(* Logix 5000 project; controller Sucrose_Main Emulate 5570 rev 20.12; software revision 20.01; part 8 of 30 *)
(* tags used below, declared in another part *)
   AI_E23_0 : REAL[8];   // Analog Input EN2T_FLX 192.168.1.23
   AI_E23_1 : REAL[8];   // Analog Input EN2T_FLX 192.168.1.23
   Alarm_ACK_Master_Timer : TIMER;
   ClearFault_Master : BOOL;
   DI_E20_0 : ALIAS FOR FLX_E20:0:I;   // Discrete Input EN2T_FLX 192.168.1.20
   DI_E20_2 : ALIAS FOR FLX_E20:2:I;   // Discrete Input EN2T_FLX 192.168.1.20
   DISCHARGE_NO_ALARM : BOOL;   // SUCROSE HEADER NO ACTIVE ALARMS FOR P_23_01_01 PATH
   DISCHARGE_NO_ALARM2 : BOOL;   // SUCROSE HEADER NO ACTIVE ALARMS FOR P_23_01_02 PATH
   DO_E20_3 : ALIAS FOR FLX_E20:3:O;   // Discrete Output EN2T_FLX 192.168.1.20
   FV230411_AOI : QSI_Flow_Valve;   // FV-23-04-11-O SUCROSE TANK #1 TO TRANSFER PUMP #1 MIX PROOF VALVE OPEN
   FV230441_AOI : QSI_Flow_Valve;   // FV-23-04-41-O SUCROSE TRANSFER PUMP #1 DISCHARGE TO FILTRATRION MIX PROOF VALVE OPEN
   FV230442_AOI : QSI_Flow_Valve;   // FV-23-04-42-O SUCROSE TRANSFER PUMP #2 DISCHARGE TO FILTRATRION MIX PROOF VALVE OPEN
   HEADER_LOW_FLOW : DINT;
   ONESHOTBITS : INT[10];
   P230401_AOI : PF525_VFD_E_ENET;   // P-23-04-01 SUCROSE TRANSFER PUMP 1
   P230402_AOI : PF525_VFD_E_ENET;   // P-23-04-02 SUCROSE TRANSFER PUMP 2
   P620101_AOI : PF525_VFD_E_ENET;   // P-62-01-01 CIP RETURN UP
   Rung_Comment : BOOL;
   SUCROSE_HEADER_NO_ALARM : BOOL;
   SUCROSE_HEADER_WATER_PURGE_GALLONS_TOTAL : DINT;
   SUCROSE_HEADER_WATER_PURGE_SP : DINT;
   Sucrose_MM_Enable : BOOL;
   SUCROSE_TANK_QUEUE_LEVEL : DINT;
   SucroseCIP_P230401_REMOTE : CIP_REMOTE;
   SucroseCIP_P230402_REMOTE : CIP_REMOTE;
   SucroseCIP_RINGMAIN_REMOTE : CIP_REMOTE;
   SucroseCIP_TK230101_REMOTE : CIP_REMOTE;
   SucroseCIP_TK230201_REMOTE : CIP_REMOTE;
   SucroseCIP_TK230301_REMOTE : CIP_REMOTE;
   SucroseDischarge : Area_Program;
   SucroseFiltration : Area_Program;
   SucroseTanks : Area_Program;
   SUROSE_HEADER_WATER_PURGE_GALS_PER_SEC : DINT;
   TK_23_01_01_LOW_LEVEL : DINT;
   TK_23_02_01_LOW_LEVEL : DINT;
   TK_23_03_01_LOW_LEVEL : DINT;
(* CIP_RemoteArea_EN2T_IO_Discrete_DO_E25_5, continued *)

ROUTINE MainRoutine   (* ladder *)
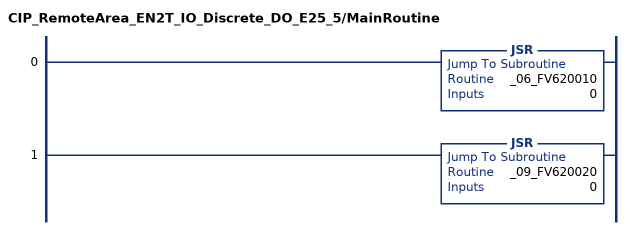
   0: JSR(_06_FV620010,0);
   1: JSR(_09_FV620020,0);
END_ROUTINE
END_PROGRAM

PROGRAM CIP_RemoteArea_EN2T_IO_Drives   (* main routine MainRoutine *)

ROUTINE E32_P620101   (* ladder *)
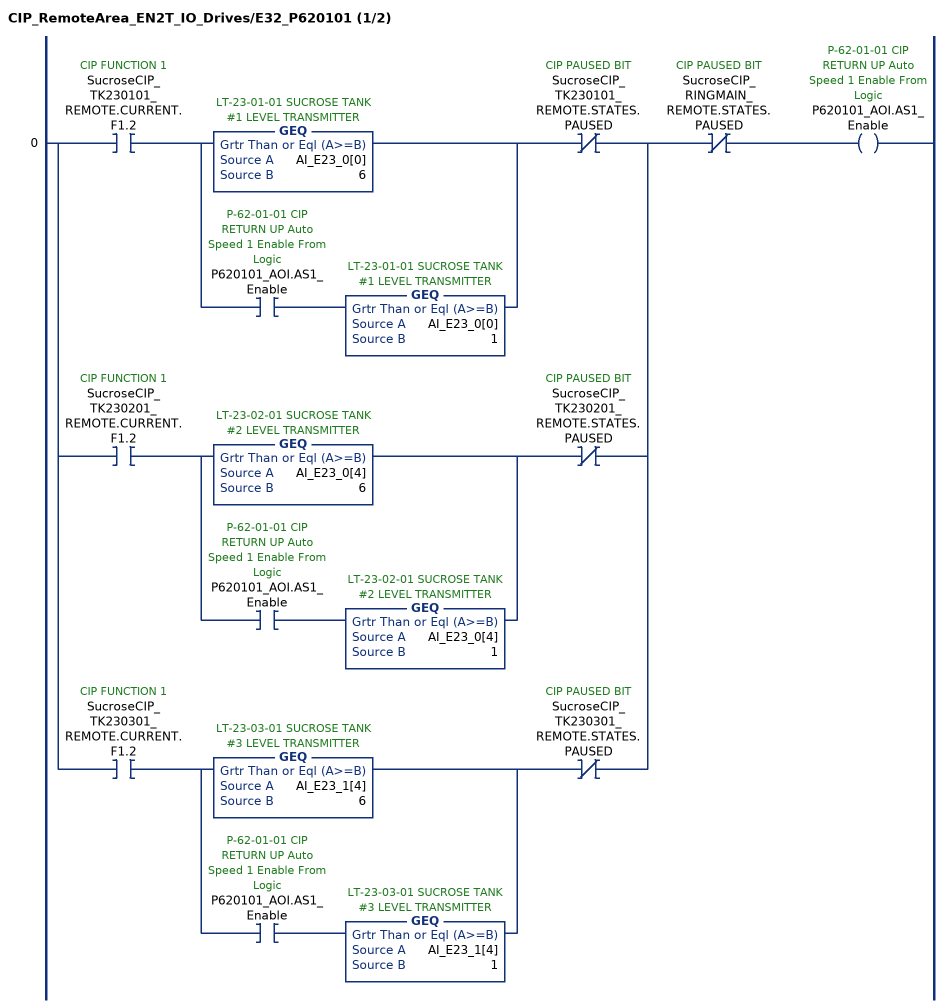
   0: [XIC(SucroseCIP_TK230101_REMOTE.CURRENT.F1.2) [GEQ(AI_E23_0[0],6) ,XIC(P620101_AOI.AS1_Enable) GEQ(AI_E23_0[0],1) ] XIO(SucroseCIP_TK230101_REMOTE.STATES.PAUSED) ,XIC(SucroseCIP_TK230201_REMOTE.CURRENT.F1.2) [GEQ(AI_E23_0[4],6) ,XIC(P620101_AOI.AS1_Enable) GEQ(AI_E23_0[4],1) ] XIO(SucroseCIP_TK230201_REMOTE.STATES.PAUSED) ,XIC(SucroseCIP_TK230301_REMOTE.CURRENT.F1.2) [GEQ(AI_E23_1[4],6) ,XIC(P620101_AOI.AS1_Enable) GEQ(AI_E23_1[4],1) ] XIO(SucroseCIP_TK230301_REMOTE.STATES.PAUSED) ]XIO(SucroseCIP_RINGMAIN_REMOTE.STATES.PAUSED)OTE(P620101_AOI.AS1_Enable);
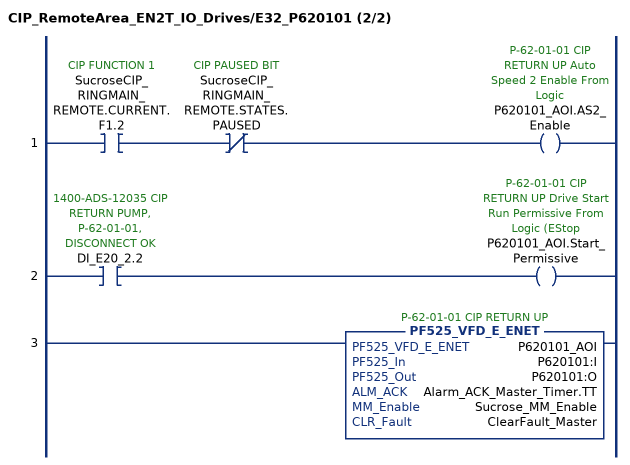
   1: XIC(SucroseCIP_RINGMAIN_REMOTE.CURRENT.F1.2)XIO(SucroseCIP_RINGMAIN_REMOTE.STATES.PAUSED)OTE(P620101_AOI.AS2_Enable);
   2: XIC(DI_E20_2.2)OTE(P620101_AOI.Start_Permissive);
   3: PF525_VFD_E_ENET(P620101_AOI,P620101:I,P620101:O,Alarm_ACK_Master_Timer.TT,Sucrose_MM_Enable,ClearFault_Master);
END_ROUTINE

ROUTINE MainRoutine   (* ladder *)
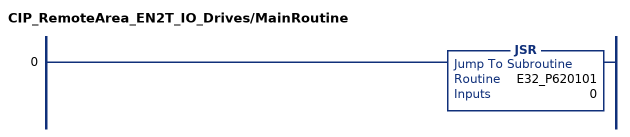
   0: JSR(E32_P620101,0);
END_ROUTINE
END_PROGRAM

PROGRAM DischargeArea_AutoLogic   (* main routine MainRoutine *)
VAR
   HEADER_HIGH_PRESSUR : DINT;
   HEADER_LOW_PRESSUR : DINT;
END_VAR

ROUTINE Alarm_Logic   (* ladder *)
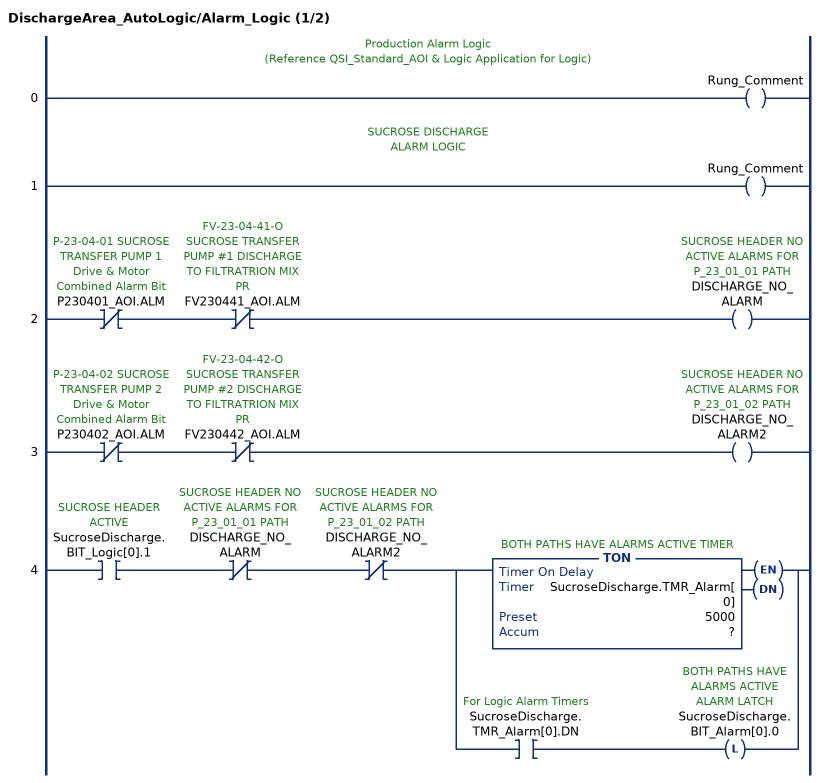
   // Production Alarm Logic
   // (Reference QSI_Standard_AOI & Logic Application for Logic)
   0: OTE(Rung_Comment);
   // SUCROSE DISCHARGE
   // ALARM LOGIC
   1: OTE(Rung_Comment);
   2: XIO(P230401_AOI.ALM)XIO(FV230441_AOI.ALM)OTE(DISCHARGE_NO_ALARM);
   3: XIO(P230402_AOI.ALM)XIO(FV230442_AOI.ALM)OTE(DISCHARGE_NO_ALARM2);
   4: XIC(SucroseDischarge.BIT_Logic[0].1)XIO(DISCHARGE_NO_ALARM)XIO(DISCHARGE_NO_ALARM2)[TON(SucroseDischarge.TMR_Alarm[0],?,?) ,XIC(SucroseDischarge.TMR_Alarm[0].DN) OTL(SucroseDischarge.BIT_Alarm[0].0) ];
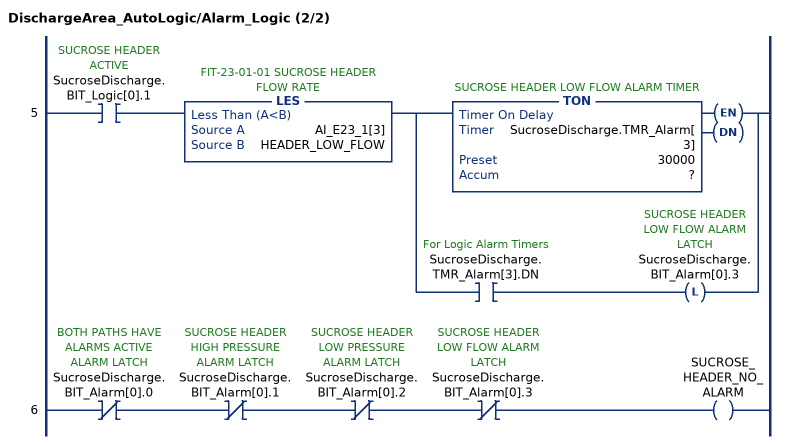
   5: XIC(SucroseDischarge.BIT_Logic[0].1)LES(AI_E23_1[3],HEADER_LOW_FLOW)[TON(SucroseDischarge.TMR_Alarm[3],?,?) ,XIC(SucroseDischarge.TMR_Alarm[3].DN) OTL(SucroseDischarge.BIT_Alarm[0].3) ];
   6: XIO(SucroseDischarge.BIT_Alarm[0].0)XIO(SucroseDischarge.BIT_Alarm[0].1)XIO(SucroseDischarge.BIT_Alarm[0].2)XIO(SucroseDischarge.BIT_Alarm[0].3)OTE(SUCROSE_HEADER_NO_ALARM);
END_ROUTINE

ROUTINE Control_Logic   (* ladder *)
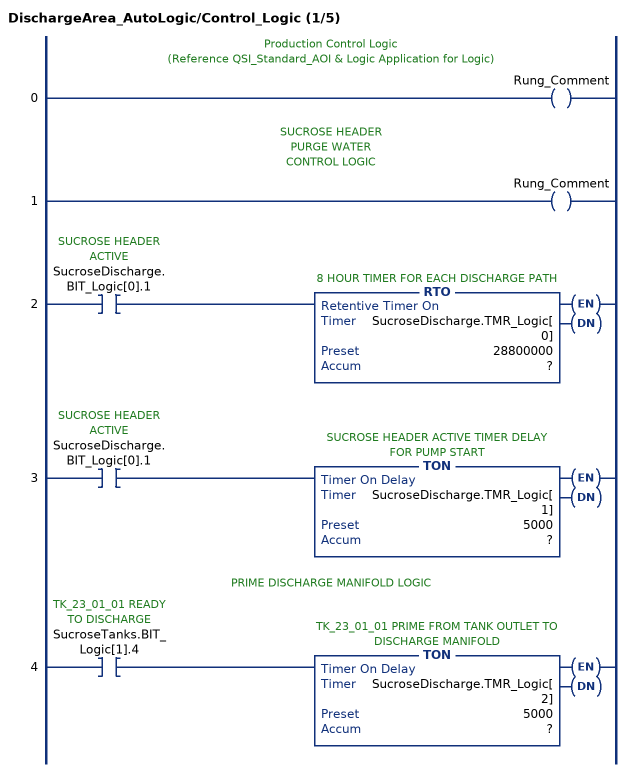
   // Production Control Logic
   // (Reference QSI_Standard_AOI & Logic Application for Logic)
   0: OTE(Rung_Comment);
   // SUCROSE HEADER
   // PURGE WATER
   // CONTROL LOGIC
   1: OTE(Rung_Comment);
   2: XIC(SucroseDischarge.BIT_Logic[0].1)RTO(SucroseDischarge.TMR_Logic[0],?,?);
   3: XIC(SucroseDischarge.BIT_Logic[0].1)TON(SucroseDischarge.TMR_Logic[1],?,?);
   // PRIME DISCHARGE MANIFOLD LOGIC
   4: XIC(SucroseTanks.BIT_Logic[1].4)TON(SucroseDischarge.TMR_Logic[2],?,?);
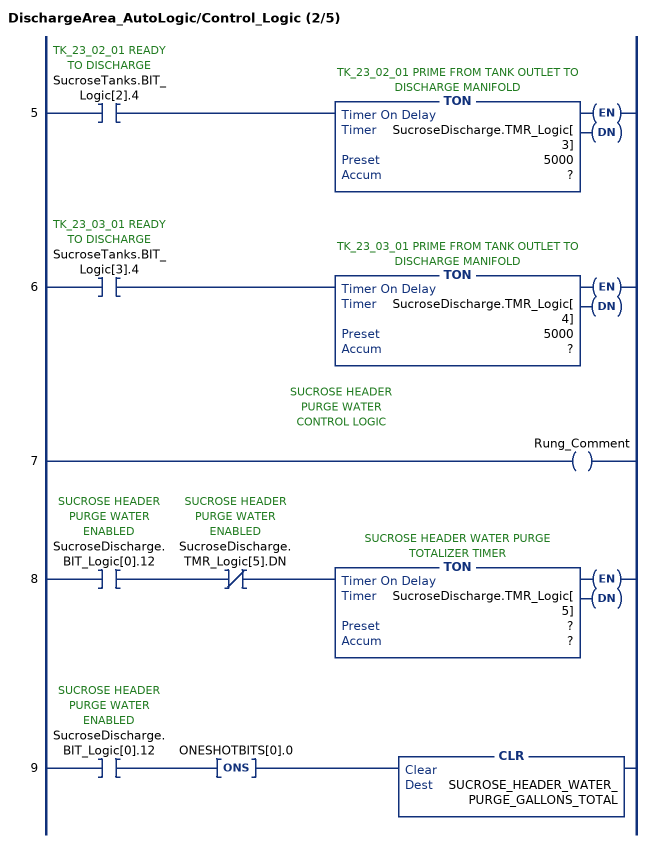
   5: XIC(SucroseTanks.BIT_Logic[2].4)TON(SucroseDischarge.TMR_Logic[3],?,?);
   6: XIC(SucroseTanks.BIT_Logic[3].4)TON(SucroseDischarge.TMR_Logic[4],?,?);
   // SUCROSE HEADER
   // PURGE WATER
   // CONTROL LOGIC
   7: OTE(Rung_Comment);
   8: XIC(SucroseDischarge.BIT_Logic[0].12)XIO(SucroseDischarge.TMR_Logic[5].DN)TON(SucroseDischarge.TMR_Logic[5],?,?);
   9: XIC(SucroseDischarge.BIT_Logic[0].12)ONS(ONESHOTBITS[0].0)CLR(SUCROSE_HEADER_WATER_PURGE_GALLONS_TOTAL);
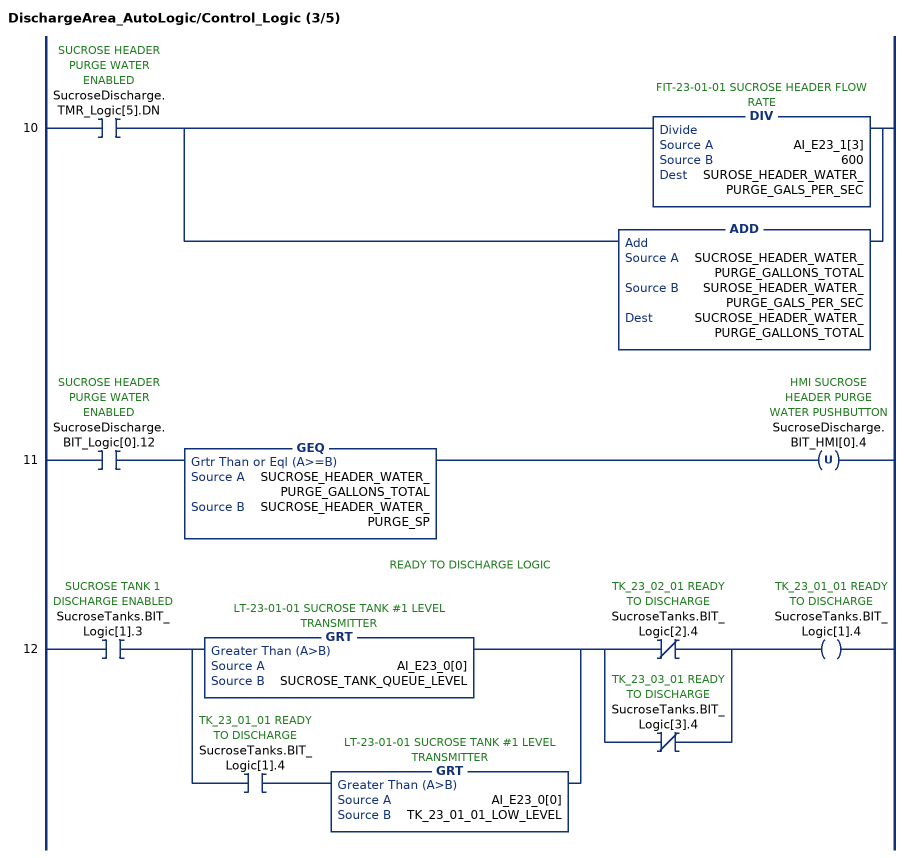
   10: XIC(SucroseDischarge.TMR_Logic[5].DN)[DIV(AI_E23_1[3],600,SUROSE_HEADER_WATER_PURGE_GALS_PER_SEC) ,ADD(SUCROSE_HEADER_WATER_PURGE_GALLONS_TOTAL,SUROSE_HEADER_WATER_PURGE_GALS_PER_SEC,SUCROSE_HEADER_WATER_PURGE_GALLONS_TOTAL) ];
   11: XIC(SucroseDischarge.BIT_Logic[0].12)GEQ(SUCROSE_HEADER_WATER_PURGE_GALLONS_TOTAL,SUCROSE_HEADER_WATER_PURGE_SP)OTU(SucroseDischarge.BIT_HMI[0].4);
   // READY TO DISCHARGE LOGIC
   12: XIC(SucroseTanks.BIT_Logic[1].3)[GRT(AI_E23_0[0],SUCROSE_TANK_QUEUE_LEVEL) ,XIC(SucroseTanks.BIT_Logic[1].4) GRT(AI_E23_0[0],TK_23_01_01_LOW_LEVEL) ][XIO(SucroseTanks.BIT_Logic[2].4) ,XIO(SucroseTanks.BIT_Logic[3].4) ]OTE(SucroseTanks.BIT_Logic[1].4);
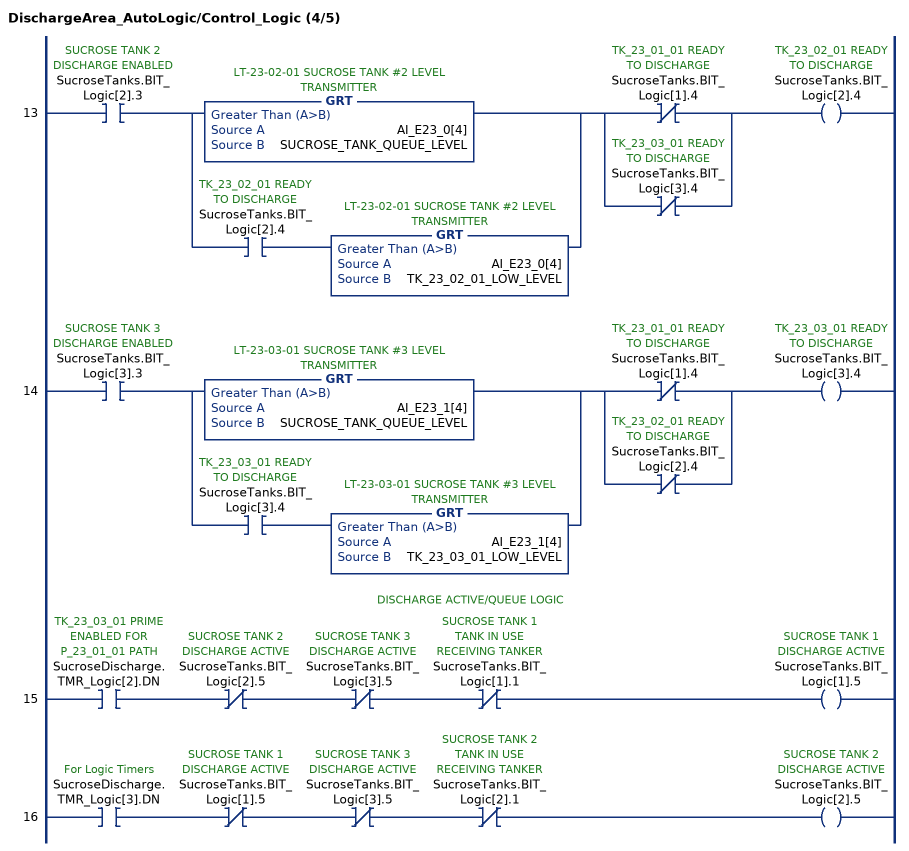
   13: XIC(SucroseTanks.BIT_Logic[2].3)[GRT(AI_E23_0[4],SUCROSE_TANK_QUEUE_LEVEL) ,XIC(SucroseTanks.BIT_Logic[2].4) GRT(AI_E23_0[4],TK_23_02_01_LOW_LEVEL) ][XIO(SucroseTanks.BIT_Logic[1].4) ,XIO(SucroseTanks.BIT_Logic[3].4) ]OTE(SucroseTanks.BIT_Logic[2].4);
   14: XIC(SucroseTanks.BIT_Logic[3].3)[GRT(AI_E23_1[4],SUCROSE_TANK_QUEUE_LEVEL) ,XIC(SucroseTanks.BIT_Logic[3].4) GRT(AI_E23_1[4],TK_23_03_01_LOW_LEVEL) ][XIO(SucroseTanks.BIT_Logic[1].4) ,XIO(SucroseTanks.BIT_Logic[2].4) ]OTE(SucroseTanks.BIT_Logic[3].4);
   // DISCHARGE ACTIVE/QUEUE LOGIC
   15: XIC(SucroseDischarge.TMR_Logic[2].DN)XIO(SucroseTanks.BIT_Logic[2].5)XIO(SucroseTanks.BIT_Logic[3].5)XIO(SucroseTanks.BIT_Logic[1].1)OTE(SucroseTanks.BIT_Logic[1].5);
   16: XIC(SucroseDischarge.TMR_Logic[3].DN)XIO(SucroseTanks.BIT_Logic[1].5)XIO(SucroseTanks.BIT_Logic[3].5)XIO(SucroseTanks.BIT_Logic[2].1)OTE(SucroseTanks.BIT_Logic[2].5);
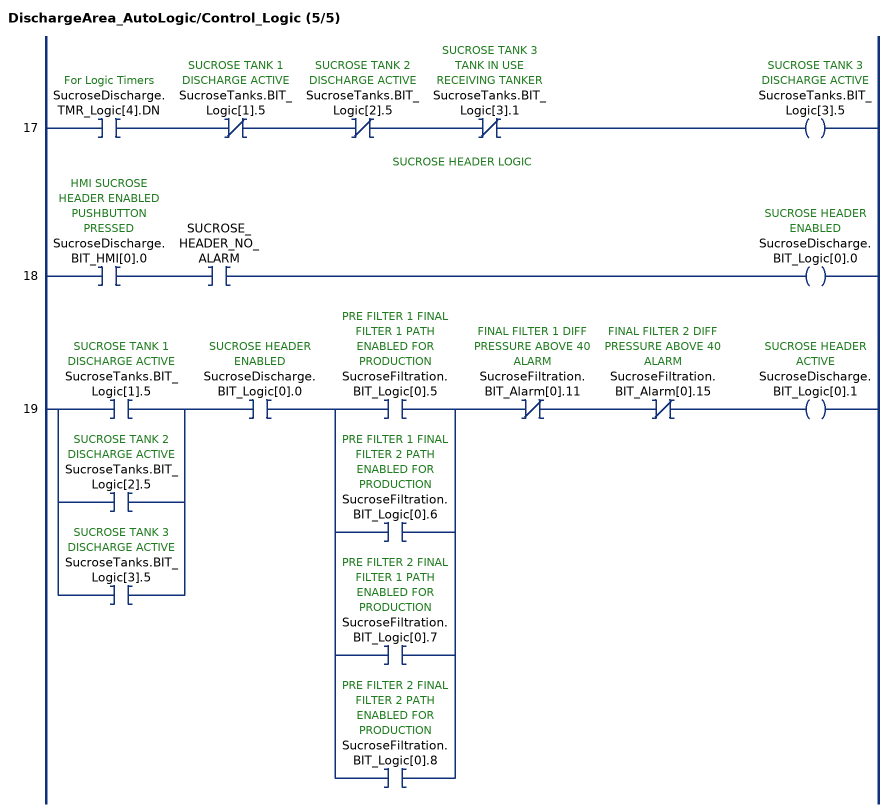
   17: XIC(SucroseDischarge.TMR_Logic[4].DN)XIO(SucroseTanks.BIT_Logic[1].5)XIO(SucroseTanks.BIT_Logic[2].5)XIO(SucroseTanks.BIT_Logic[3].1)OTE(SucroseTanks.BIT_Logic[3].5);
   // SUCROSE HEADER LOGIC
   18: XIC(SucroseDischarge.BIT_HMI[0].0)XIC(SUCROSE_HEADER_NO_ALARM)OTE(SucroseDischarge.BIT_Logic[0].0);
   19: [XIC(SucroseTanks.BIT_Logic[1].5) ,XIC(SucroseTanks.BIT_Logic[2].5) ,XIC(SucroseTanks.BIT_Logic[3].5) ]XIC(SucroseDischarge.BIT_Logic[0].0)[XIC(SucroseFiltration.BIT_Logic[0].5) ,XIC(SucroseFiltration.BIT_Logic[0].6) ,XIC(SucroseFiltration.BIT_Logic[0].7) ,XIC(SucroseFiltration.BIT_Logic[0].8) ]XIO(SucroseFiltration.BIT_Alarm[0].11)XIO(SucroseFiltration.BIT_Alarm[0].15)OTE(SucroseDischarge.BIT_Logic[0].1);
END_ROUTINE

ROUTINE Enable_Logic   (* ladder *)
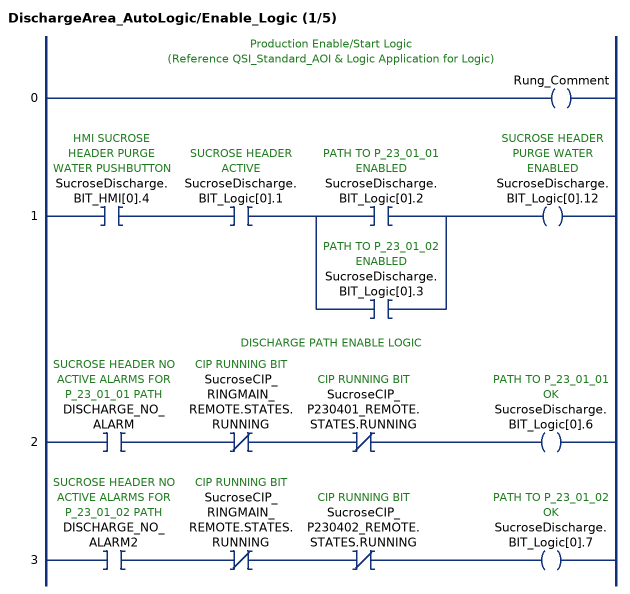
   // Production Enable/Start Logic
   // (Reference QSI_Standard_AOI & Logic Application for Logic)
   0: OTE(Rung_Comment);
   1: XIC(SucroseDischarge.BIT_HMI[0].4)XIC(SucroseDischarge.BIT_Logic[0].1)[XIC(SucroseDischarge.BIT_Logic[0].2) ,XIC(SucroseDischarge.BIT_Logic[0].3) ]OTE(SucroseDischarge.BIT_Logic[0].12);
   // DISCHARGE PATH ENABLE LOGIC
   2: XIC(DISCHARGE_NO_ALARM)XIO(SucroseCIP_RINGMAIN_REMOTE.STATES.RUNNING)XIO(SucroseCIP_P230401_REMOTE.STATES.RUNNING)OTE(SucroseDischarge.BIT_Logic[0].6);
   3: XIC(DISCHARGE_NO_ALARM2)XIO(SucroseCIP_RINGMAIN_REMOTE.STATES.RUNNING)XIO(SucroseCIP_P230402_REMOTE.STATES.RUNNING)OTE(SucroseDischarge.BIT_Logic[0].7);
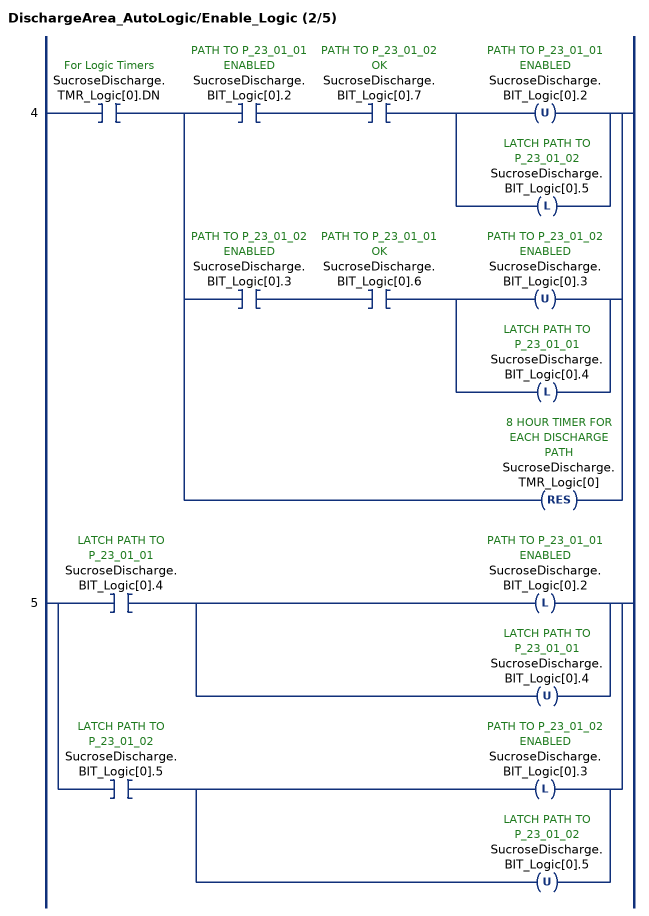
   4: XIC(SucroseDischarge.TMR_Logic[0].DN)[XIC(SucroseDischarge.BIT_Logic[0].2) XIC(SucroseDischarge.BIT_Logic[0].7) [OTU(SucroseDischarge.BIT_Logic[0].2) ,OTL(SucroseDischarge.BIT_Logic[0].5) ] ,XIC(SucroseDischarge.BIT_Logic[0].3) XIC(SucroseDischarge.BIT_Logic[0].6) [OTU(SucroseDischarge.BIT_Logic[0].3) ,OTL(SucroseDischarge.BIT_Logic[0].4) ] ,RES(SucroseDischarge.TMR_Logic[0]) ];
   5: [XIC(SucroseDischarge.BIT_Logic[0].4) [OTL(SucroseDischarge.BIT_Logic[0].2) ,OTU(SucroseDischarge.BIT_Logic[0].4) ] ,XIC(SucroseDischarge.BIT_Logic[0].5) [OTL(SucroseDischarge.BIT_Logic[0].3) ,OTU(SucroseDischarge.BIT_Logic[0].5) ] ];
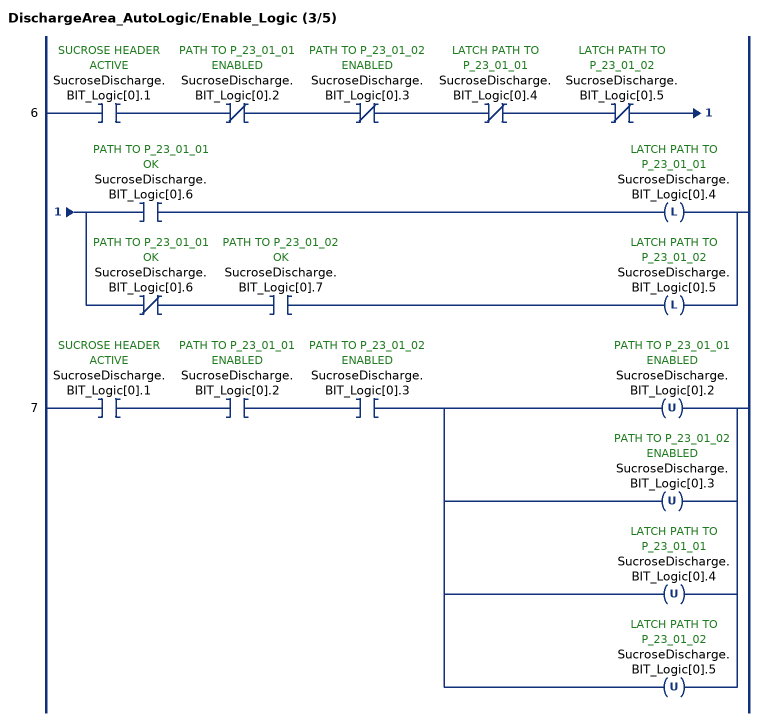
   6: XIC(SucroseDischarge.BIT_Logic[0].1)XIO(SucroseDischarge.BIT_Logic[0].2)XIO(SucroseDischarge.BIT_Logic[0].3)XIO(SucroseDischarge.BIT_Logic[0].4)XIO(SucroseDischarge.BIT_Logic[0].5)[XIC(SucroseDischarge.BIT_Logic[0].6) OTL(SucroseDischarge.BIT_Logic[0].4) ,XIO(SucroseDischarge.BIT_Logic[0].6) XIC(SucroseDischarge.BIT_Logic[0].7) OTL(SucroseDischarge.BIT_Logic[0].5) ];
   7: XIC(SucroseDischarge.BIT_Logic[0].1)XIC(SucroseDischarge.BIT_Logic[0].2)XIC(SucroseDischarge.BIT_Logic[0].3)[OTU(SucroseDischarge.BIT_Logic[0].2) ,OTU(SucroseDischarge.BIT_Logic[0].3) ,OTU(SucroseDischarge.BIT_Logic[0].4) ,OTU(SucroseDischarge.BIT_Logic[0].5) ];
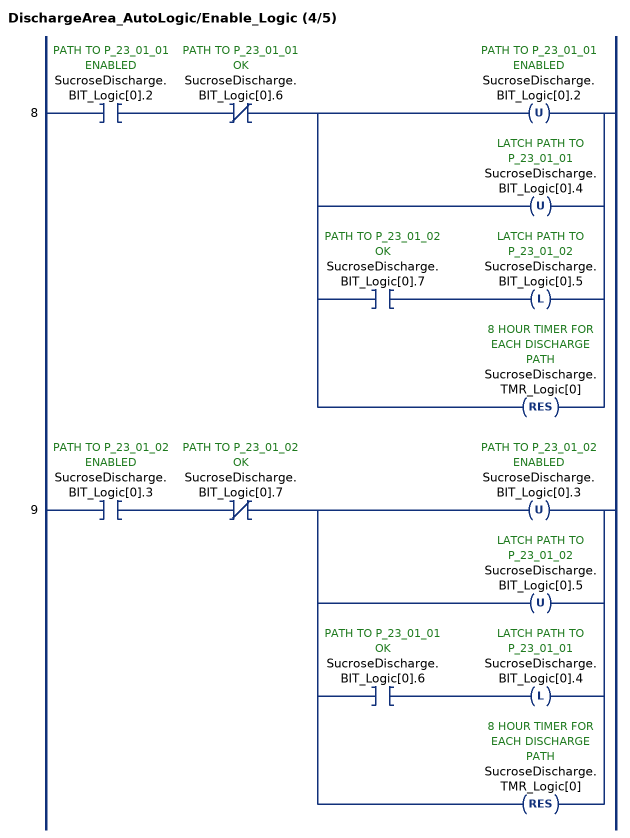
   8: XIC(SucroseDischarge.BIT_Logic[0].2)XIO(SucroseDischarge.BIT_Logic[0].6)[OTU(SucroseDischarge.BIT_Logic[0].2) ,OTU(SucroseDischarge.BIT_Logic[0].4) ,XIC(SucroseDischarge.BIT_Logic[0].7) OTL(SucroseDischarge.BIT_Logic[0].5) ,RES(SucroseDischarge.TMR_Logic[0]) ];
   9: XIC(SucroseDischarge.BIT_Logic[0].3)XIO(SucroseDischarge.BIT_Logic[0].7)[OTU(SucroseDischarge.BIT_Logic[0].3) ,OTU(SucroseDischarge.BIT_Logic[0].5) ,XIC(SucroseDischarge.BIT_Logic[0].6) OTL(SucroseDischarge.BIT_Logic[0].4) ,RES(SucroseDischarge.TMR_Logic[0]) ];
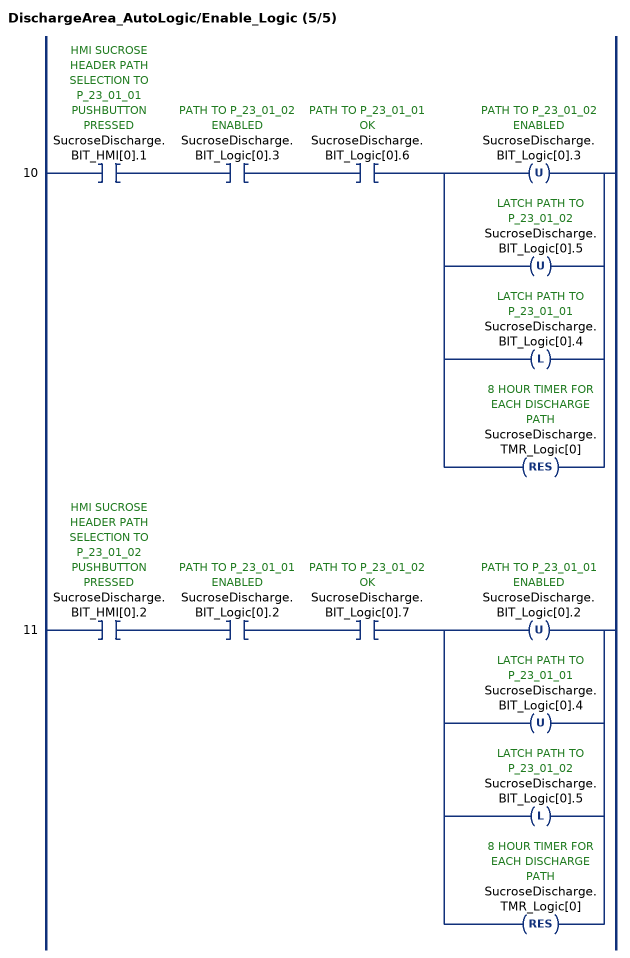
   10: XIC(SucroseDischarge.BIT_HMI[0].1)XIC(SucroseDischarge.BIT_Logic[0].3)XIC(SucroseDischarge.BIT_Logic[0].6)[OTU(SucroseDischarge.BIT_Logic[0].3) ,OTU(SucroseDischarge.BIT_Logic[0].5) ,OTL(SucroseDischarge.BIT_Logic[0].4) ,RES(SucroseDischarge.TMR_Logic[0]) ];
   11: XIC(SucroseDischarge.BIT_HMI[0].2)XIC(SucroseDischarge.BIT_Logic[0].2)XIC(SucroseDischarge.BIT_Logic[0].7)[OTU(SucroseDischarge.BIT_Logic[0].2) ,OTU(SucroseDischarge.BIT_Logic[0].4) ,OTL(SucroseDischarge.BIT_Logic[0].5) ,RES(SucroseDischarge.TMR_Logic[0]) ];
END_ROUTINE

ROUTINE MainRoutine   (* ladder *)
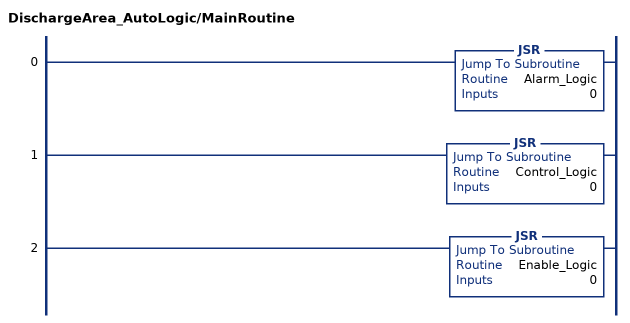
   0: JSR(Alarm_Logic,0);
   1: JSR(Control_Logic,0);
   2: JSR(Enable_Logic,0);
END_ROUTINE
END_PROGRAM

PROGRAM DischargeArea_EN2T_IO_Discrete_DO_E20_3   (* main routine MainRoutine *)

ROUTINE _00_FV230411   (* ladder *)
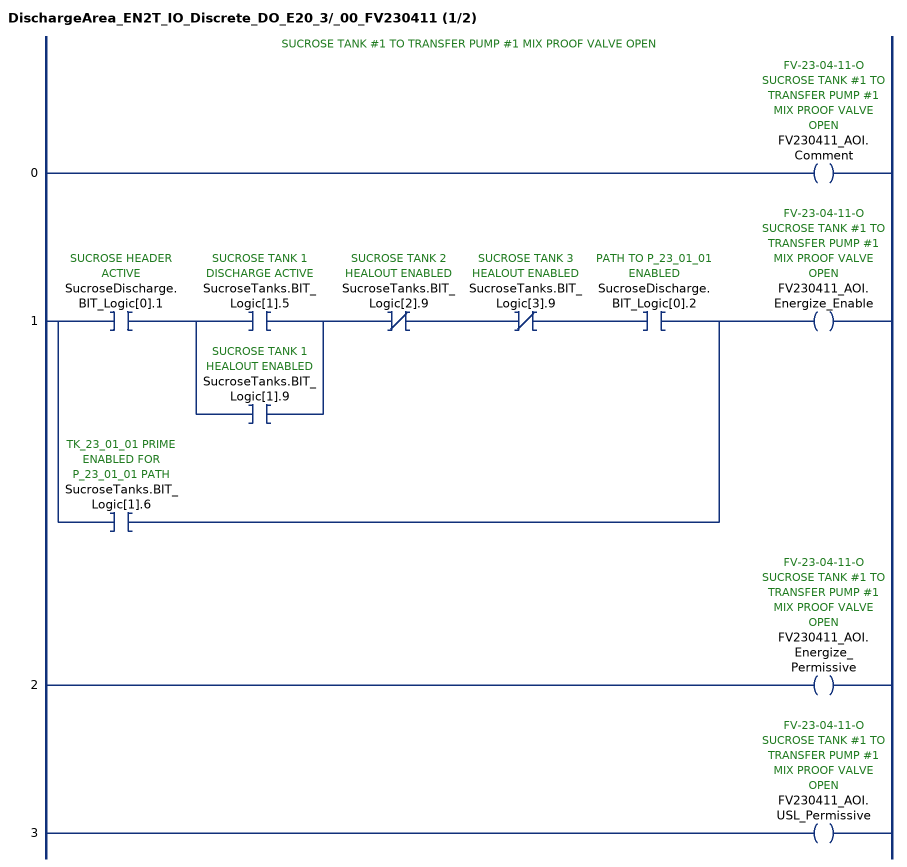
   // SUCROSE TANK #1 TO TRANSFER PUMP #1 MIX PROOF VALVE OPEN
   0: OTE(FV230411_AOI.Comment);
   1: [XIC(SucroseDischarge.BIT_Logic[0].1) [XIC(SucroseTanks.BIT_Logic[1].5) ,XIC(SucroseTanks.BIT_Logic[1].9) ] XIO(SucroseTanks.BIT_Logic[2].9) XIO(SucroseTanks.BIT_Logic[3].9) XIC(SucroseDischarge.BIT_Logic[0].2) ,XIC(SucroseTanks.BIT_Logic[1].6) ]OTE(FV230411_AOI.Energize_Enable);
   2: OTE(FV230411_AOI.Energize_Permissive);
   3: OTE(FV230411_AOI.USL_Permissive);
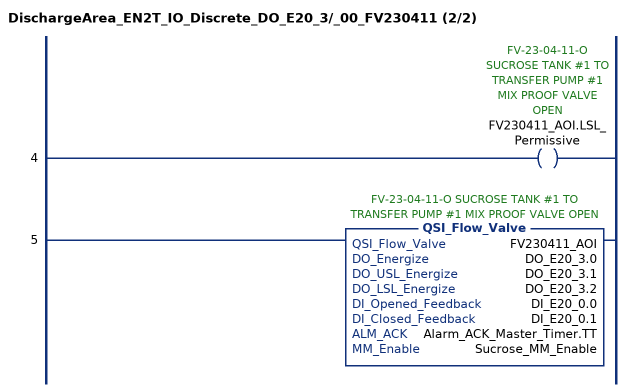
   4: OTE(FV230411_AOI.LSL_Permissive);
   5: QSI_Flow_Valve(FV230411_AOI,DO_E20_3.0,DO_E20_3.1,DO_E20_3.2,DI_E20_0.0,DI_E20_0.1,Alarm_ACK_Master_Timer.TT,Sucrose_MM_Enable);
END_ROUTINE
